// TwinCAT 3 PLC project Simulation
// ProgramVersion: 3.1.4026.26
// libraries:
//   Tc2_Standard, 3.4.7.0 (Beckhoff Automation GmbH)
//   Tc2_System, 3.10.2.0 (Beckhoff Automation GmbH)
//   [TcForge], 2.0.0.0 (Home)
//   [TcForgeExample], 2.0.0.0 (Home)
// project tree:
//   Simulation/ FB_ArchitectureFixture.TcPOU, PRG_OwnershipWitness.TcPOU, OwnershipWitness.TcTTO, FB_LifecycleFixture.TcPOU, MAIN.TcPOU, Simulation.TcTTO
// (motion and I/O tree: see PLC project tcforge)
// real-time tasks:
//   TASK OwnershipWitness: cycle T#10ms, priority 4, ADS port 353
//   TASK Simulation: cycle T#10ms, priority 3, ADS port 352

CONFIGURATION Simulation
    RESOURCE PLC ON TwinCAT3
        TASK OwnershipWitness(INTERVAL := T#10ms, PRIORITY := 4);
        TASK Simulation(INTERVAL := T#10ms, PRIORITY := 3);
        PROGRAM PRG_OwnershipWitness WITH OwnershipWitness : PRG_OwnershipWitness;
        PROGRAM MAIN WITH Simulation : MAIN;
    END_RESOURCE
END_CONFIGURATION

// ---- Simulation/PRG_OwnershipWitness.TcPOU
PROGRAM PRG_OwnershipWitness
VAR taskIndex : DINT; cycles : ULINT; END_VAR

taskIndex := Tc2_System.GETCURTASKINDEXEX(); cycles := cycles + 1;
// The owner deliberately yields this instance until this one conflicting call is complete.
// This proves deterministic ownership detection, not arbitrary cross-task memory safety.
IF MAIN.ownershipHandoff AND NOT MAIN.ownershipWitnessDone THEN
    MAIN.sharedOutput();
    MAIN.ownershipWitnessTask := taskIndex;
    MAIN.ownershipWitnessDone := TRUE;
END_IF;

END_PROGRAM

// ---- Simulation/MAIN.TcPOU
PROGRAM MAIN
VAR_INPUT
    ownershipWitnessDone : BOOL;
    ownershipWitnessTask : DINT;
END_VAR
VAR
    simulation : FB_SimulationBridge; lifecycle : FB_LifecycleFixture;
    architecture : FB_ArchitectureFixture;
    sharedOutput : TcForge.FB_DigitalOutput;
    ownershipKick, ownershipHandoff : BOOL;
    ownershipPhase : UINT;
    ownershipOwnerTask : DINT;
    ownershipInitialAdmission, ownershipInitialResult, ownershipQueued,
        ownershipCancelled, ownershipRejected : TcForge.E_RpcMethodResponse;
    ownershipInitiallyOn, ownershipFinalOutput : BOOL;
END_VAR

simulation();
lifecycle();
architecture();
IF NOT ownershipHandoff OR ownershipWitnessDone THEN sharedOutput(); END_IF;
CASE ownershipPhase OF
0:
    IF ownershipKick THEN
        ownershipOwnerTask := Tc2_System.GETCURTASKINDEXEX();
        ownershipInitialAdmission := sharedOutput.OperatorSetOn(requestId := 101);
        ownershipPhase := 1;
    END_IF;
1:
    ownershipInitialResult := sharedOutput.OperatorCommandResult(requestId := 101);
    IF ownershipInitialResult = TcForge.E_RpcMethodResponse.ACCEPTED AND sharedOutput.outSignal THEN
        ownershipInitiallyOn := TRUE; sharedOutput.ForceSafe(); ownershipPhase := 2;
    END_IF;
2:
    IF NOT sharedOutput.outSignal THEN
        ownershipQueued := sharedOutput.OperatorSetOn(requestId := 102);
        ownershipHandoff := TRUE; ownershipPhase := 3;
    END_IF;
3:
    IF ownershipWitnessDone THEN
        ownershipCancelled := sharedOutput.OperatorCommandResult(requestId := 102);
        ownershipRejected := sharedOutput.OperatorSetOn(requestId := 103);
        ownershipFinalOutput := sharedOutput.outSignal; ownershipPhase := 4;
    END_IF;
END_CASE;

END_PROGRAM

// ---- Simulation/FB_LifecycleFixture.TcPOU
// Standalone qualification fixture: no physical IO mapping, no RPC methods.
// ADS client writes commandCode first, then a strictly increasing commandSequence.
// Read completedSequence before issuing another command. One owner task calls once/scan.
// These PERSISTENT declarations require actual runtime validation; they promise no
// sudden-power-loss durability. No automatic writes to the persistent image are requested.
FUNCTION_BLOCK FB_LifecycleFixture
VAR_INPUT
    commandCode : UINT;
    commandSequence : UDINT;
END_VAR
VAR_OUTPUT
    completedSequence : UDINT;
    commandAccepted : BOOL;
    initialized : BOOL;
    cycles : ULINT;
    markerAtInitialization : UINT;
    bootDataLoadedAtInitialization : BOOL;
    oldBootDataAtInitialization : BOOL;
    onlineChangeCount : UDINT;
    defaultOutput : BOOL;
    defaultInhibited : BOOL;
    restoreOutput : BOOL;
    restoreInhibited : BOOL;
    analogRaw : REAL;
    analogInhibited : BOOL;
    alarmActive : BOOL;
    alarmLatched : BOOL;
    alarmAcked : BOOL;
    diagnosticFaulted : BOOL;
    diagnosticLastFault : DINT;
    lastDefaultResponse : TcForge.E_RpcMethodResponse;
    lastRestoreResponse : TcForge.E_RpcMethodResponse;
    lastAnalogResponse : TcForge.E_RpcMethodResponse;
END_VAR
VAR PERSISTENT
    applicationMarker : UINT;
    // Application-owned configuration is restored before device first observation.
    defaultConfig : TcForge.ST_DigitalOutput_Cfg;
    restoreConfig : TcForge.ST_DigitalOutput_Cfg := (restoreCommandOnRestart := TRUE, invert := TRUE);
    analogConfig : TcForge.ST_AnalogOutput_Cfg := (restoreCommandOnRestart := TRUE, useRawValue := TRUE, safeRaw := 17.0);
    alarmConfig : TcForge.ST_AlarmSimple_Cfg := (common := (bEnable := TRUE, bRequireAck := TRUE, eSeverity := TcForge.E_AlarmSeverity.WARNING));
END_VAR
VAR
    defaultDevice : TcForge.FB_DigitalOutput;
    restoreDevice : TcForge.FB_DigitalOutput;
    analogDevice : TcForge.FB_AnalogOutput;
    alarmDevice : TcForge.FB_AlarmSimple;
    diagnosticDevice : TcForge.FB_TwoPosActuator;
    seedPulse : BOOL;
    observedSequence : UDINT;
    observedCode : UINT;
END_VAR

IF NOT initialized THEN
    markerAtInitialization := applicationMarker;
    bootDataLoadedAtInitialization := TwinCAT_SystemInfoVarList._AppInfo.BootDataLoaded;
    oldBootDataAtInitialization := TwinCAT_SystemInfoVarList._AppInfo.OldBootData;
    initialized := TRUE;
END_IF;
cycles := cycles + 1;
onlineChangeCount := TwinCAT_SystemInfoVarList._AppInfo.OnlineChangeCnt;
defaultDevice.cfg := defaultConfig;
restoreDevice.cfg := restoreConfig;
analogDevice.cfg := analogConfig;
alarmDevice.cfg := alarmConfig;
seedPulse := FALSE;
observedSequence := commandSequence;
observedCode := commandCode;
IF observedSequence > completedSequence THEN
    commandAccepted := TRUE;
    CASE observedCode OF
    1: // Seed diagnostic history, an unacknowledged latch and real operating commands.
        applicationMarker := UINT#49374;
        lastDefaultResponse := defaultDevice.SetOn();
        lastRestoreResponse := restoreDevice.SetOff(); // Inverted electrical TRUE is intentional.
        lastAnalogResponse := analogDevice.SetValue(rValue := 42.0);
        seedPulse := TRUE;
    2: // Invalidate saved output intent; diagnostic/alarm history is deliberately untouched.
        lastDefaultResponse := defaultDevice.ForceSafe();
        lastRestoreResponse := restoreDevice.ForceSafe();
        lastAnalogResponse := analogDevice.ForceSafe();
    3: // Reset outputs/active diagnostic fault; preserve history and the alarm latch.
        lastDefaultResponse := defaultDevice.Reset();
        lastRestoreResponse := restoreDevice.Reset();
        lastAnalogResponse := analogDevice.Reset();
        diagnosticDevice.Reset();
    4: // Acknowledge while this scan supplies valid clear evidence.
        alarmDevice.Ack();
    ELSE
        commandAccepted := FALSE;
    END_CASE;
END_IF;
defaultDevice();
restoreDevice();
analogDevice();
alarmDevice(inpValid := TRUE, inpActive := seedPulse);
diagnosticDevice(inAdvanced := seedPulse, inRetracted := seedPulse);
defaultOutput := defaultDevice.outSignal;
defaultInhibited := defaultDevice.sts.outputInhibited;
restoreOutput := restoreDevice.outSignal;
restoreInhibited := restoreDevice.sts.outputInhibited;
analogRaw := analogDevice.sts.rawReal;
analogInhibited := analogDevice.sts.outputInhibited;
alarmActive := alarmDevice.sts.active;
alarmLatched := alarmDevice.sts.latched;
alarmAcked := alarmDevice.sts.acked;
diagnosticFaulted := diagnosticDevice.IsFaulted();
diagnosticLastFault := diagnosticDevice.sts.header.lastFaultCode;
// Publish command completion only after owner-task evaluation and output publication.
IF observedSequence > completedSequence THEN completedSequence := observedSequence; END_IF;

END_FUNCTION_BLOCK

// ---- Simulation/FB_ArchitectureFixture.TcPOU
// Dedicated unmapped bench fixture. Commands/sensors are driven only by the qualification runner.
FUNCTION_BLOCK FB_ArchitectureFixture
VAR_INPUT
    enabled : BOOL;
    homeCommand, startCommand : E_ReferenceCommand;
    advanced : BOOL;
    retracted : BOOL := TRUE;
END_VAR
VAR_OUTPUT
    homeMachine, startMachine : FB_ReferenceMachine;
    cycles : ULINT;
    owner : DINT;
    gapCount, gapCycleDelta : UDINT;
    gapHomeResponse, gapStartResponse : TcForge.E_RpcMethodResponse;
    gapHomeAdvance, gapHomeRetract, gapStartAdvance, gapStartRetract : BOOL;
    gapHomeInhibited, gapStartInhibited : BOOL;
END_VAR
VAR known, gap : BOOL; current, previous, expected : UDINT; END_VAR

IF NOT enabled THEN RETURN; END_IF;
owner := Tc2_System.GETCURTASKINDEXEX();
IF owner <= 0 THEN RETURN; END_IF;
current := TwinCAT_SystemInfoVarList._TaskInfo[owner].CycleCount;
IF previous = UDINT#16#FFFFFFFF THEN expected := 0; ELSE expected := previous + 1; END_IF;
gap := known AND current <> previous AND current <> expected;
// No synthetic counter injection and no IO watchdog: this isolates real execution-gap protection.
homeMachine(command := homeCommand, recoverOnOnlineChange := FALSE,
    inAdvanced := advanced, inRetracted := retracted,
    inputQuality := TcForge.E_IO_Quality.GOOD, outputQuality := TcForge.E_IO_Quality.GOOD,
    shutdownConfirmed := TRUE, shutdownQuality := TcForge.E_IO_Quality.GOOD);
startMachine(command := startCommand, recoverOnOnlineChange := FALSE,
    inAdvanced := advanced, inRetracted := retracted,
    inputQuality := TcForge.E_IO_Quality.GOOD, outputQuality := TcForge.E_IO_Quality.GOOD,
    shutdownConfirmed := TRUE, shutdownQuality := TcForge.E_IO_Quality.GOOD);
IF gap THEN
    gapCount := gapCount + 1; gapCycleDelta := current - previous;
    gapHomeResponse := homeMachine.lastResponse; gapStartResponse := startMachine.lastResponse;
    gapHomeAdvance := homeMachine.outAdvance; gapHomeRetract := homeMachine.outRetract;
    gapStartAdvance := startMachine.outAdvance; gapStartRetract := startMachine.outRetract;
    gapHomeInhibited := homeMachine.outputsInhibited; gapStartInhibited := startMachine.outputsInhibited;
END_IF;
known := TRUE; previous := current; cycles := cycles + 1;

END_FUNCTION_BLOCK
